// Mitsubishi GX Works2 project: mitsu_SCADA_PLC_v6.1   PLC: FX1N/FX1NC

PROGRAM MAIN
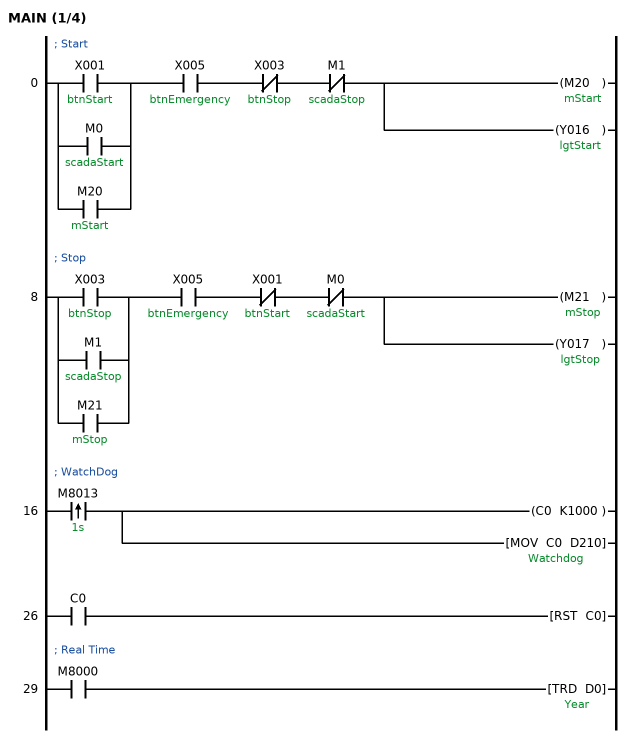
; Start
0     LD      X001  ; btnStart
      OR      M0  ; scadaStart
      OR      M20  ; mStart
      AND     X005  ; btnEmergency
      ANI     X003  ; btnStop
      ANI     M1  ; scadaStop
      OUT     M20  ; mStart
      OUT     Y016  ; lgtStart
; Stop
8     LD      X003  ; btnStop
      OR      M1  ; scadaStop
      OR      M21  ; mStop
      AND     X005  ; btnEmergency
      ANI     X001  ; btnStart
      ANI     M0  ; scadaStart
      OUT     M21  ; mStop
      OUT     Y017  ; lgtStop
; WatchDog
16    LDP     M8013  ; 1s
      OUT     C0 K1000
      MOV     C0 D210  ; Watchdog
26    LD      C0
      RST     C0
; Real Time
29    LD      M8000
      TRD     D0  ; Year
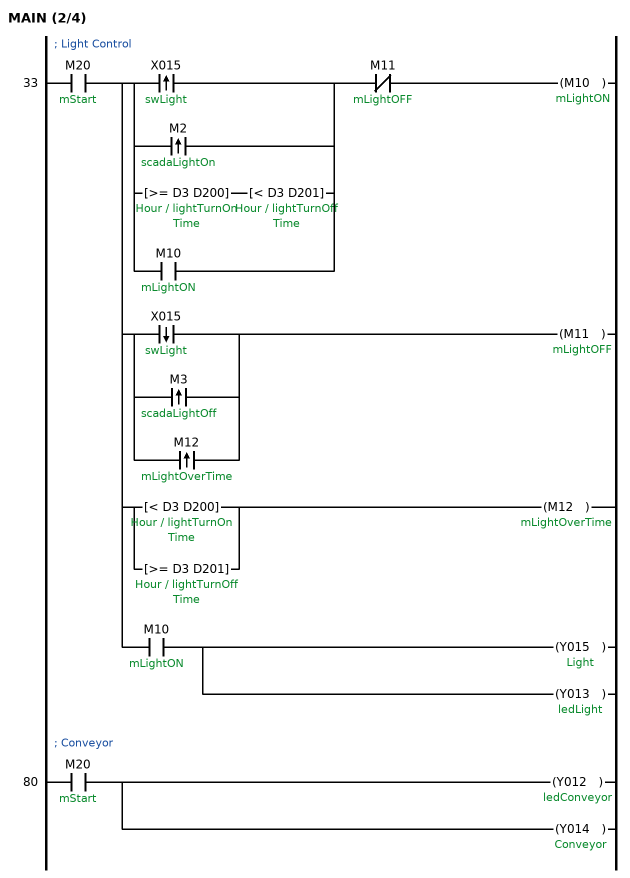
; Light Control
33    LD      M20  ; mStart
      MPS
      LDP     X015  ; swLight
      ORP     M2  ; scadaLightOn
      LD>=    D3 D200  ; Hour / lightTurnOnTime
      AND<    D3 D201  ; Hour / lightTurnOffTime
      ORB
      OR      M10  ; mLightON
      ANB
      ANI     M11  ; mLightOFF
      OUT     M10  ; mLightON
      MRD
      LDF     X015  ; swLight
      ORP     M3  ; scadaLightOff
      ORP     M12  ; mLightOverTime
      ANB
      OUT     M11  ; mLightOFF
      MRD
      LD<     D3 D200  ; Hour / lightTurnOnTime
      OR>=    D3 D201  ; Hour / lightTurnOffTime
      ANB
      OUT     M12  ; mLightOverTime
      MPP
      AND     M10  ; mLightON
      OUT     Y015  ; Light
      OUT     Y013  ; ledLight
; Conveyor
80    LD      M20  ; mStart
      OUT     Y012  ; ledConveyor
      OUT     Y014  ; Conveyor
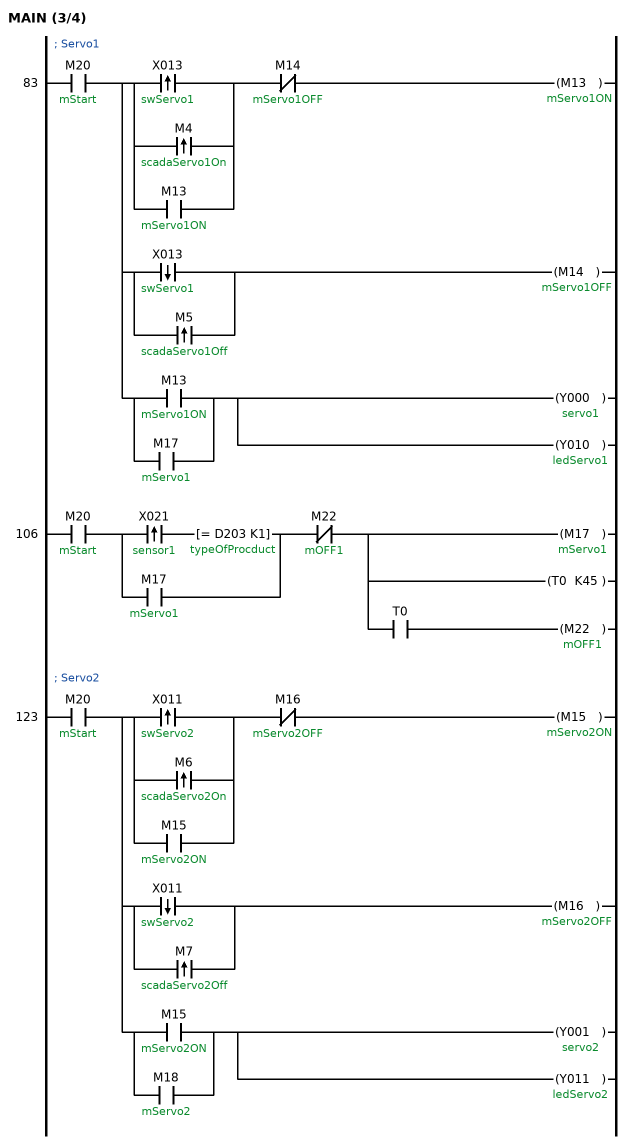
; Servo1
83    LD      M20  ; mStart
      MPS
      LDP     X013  ; swServo1
      ORP     M4  ; scadaServo1On
      OR      M13  ; mServo1ON
      ANB
      ANI     M14  ; mServo1OFF
      OUT     M13  ; mServo1ON
      MRD
      LDF     X013  ; swServo1
      ORP     M5  ; scadaServo1Off
      ANB
      OUT     M14  ; mServo1OFF
      MPP
      LD      M13  ; mServo1ON
      OR      M17  ; mServo1
      ANB
      OUT     Y000  ; servo1
      OUT     Y010  ; ledServo1
106   LD      M20  ; mStart
      LDP     X021  ; sensor1
      AND=    D203 K1  ; typeOfProcduct
      OR      M17  ; mServo1
      ANB
      ANI     M22  ; mOFF1
      OUT     M17  ; mServo1
      OUT     T0 K45
      AND     T0
      OUT     M22  ; mOFF1
; Servo2
123   LD      M20  ; mStart
      MPS
      LDP     X011  ; swServo2
      ORP     M6  ; scadaServo2On
      OR      M15  ; mServo2ON
      ANB
      ANI     M16  ; mServo2OFF
      OUT     M15  ; mServo2ON
      MRD
      LDF     X011  ; swServo2
      ORP     M7  ; scadaServo2Off
      ANB
      OUT     M16  ; mServo2OFF
      MPP
      LD      M15  ; mServo2ON
      OR      M18  ; mServo2
      ANB
      OUT     Y001  ; servo2
      OUT     Y011  ; ledServo2
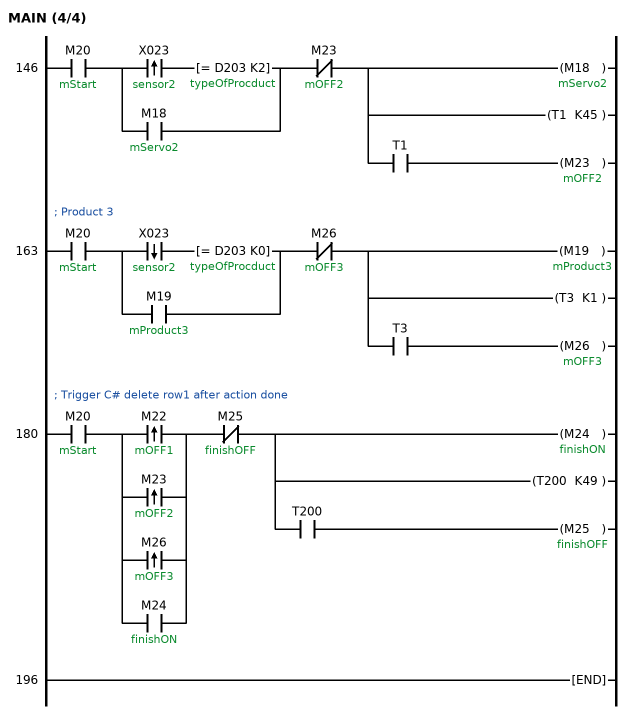
146   LD      M20  ; mStart
      LDP     X023  ; sensor2
      AND=    D203 K2  ; typeOfProcduct
      OR      M18  ; mServo2
      ANB
      ANI     M23  ; mOFF2
      OUT     M18  ; mServo2
      OUT     T1 K45
      AND     T1
      OUT     M23  ; mOFF2
; Product 3
163   LD      M20  ; mStart
      LDF     X023  ; sensor2
      AND=    D203 K0  ; typeOfProcduct
      OR      M19  ; mProduct3
      ANB
      ANI     M26  ; mOFF3
      OUT     M19  ; mProduct3
      OUT     T3 K1
      AND     T3
      OUT     M26  ; mOFF3
; Trigger C# delete row1 after action done
180   LD      M20  ; mStart
      LDP     M22  ; mOFF1
      ORP     M23  ; mOFF2
      ORP     M26  ; mOFF3
      OR      M24  ; finishON
      ANB
      ANI     M25  ; finishOFF
      OUT     M24  ; finishON
      OUT     T200 K49
      AND     T200
      OUT     M25  ; finishOFF
196   END
END_PROGRAM

// device comments not shown above
M50  ; temp_0
M51  ; temp_1
M52  ; temp_2
M53  ; temp_3
M54  ; temp_4
M55  ; temp_5
D1  ; Month
D2  ; Day
D4  ; Minute
D5  ; Second
D6  ; Date
D202  ; temperature
